// Mitsubishi GX Works2 project: 525252   PLC: Q02/Q02H

PROGRAM MAIN
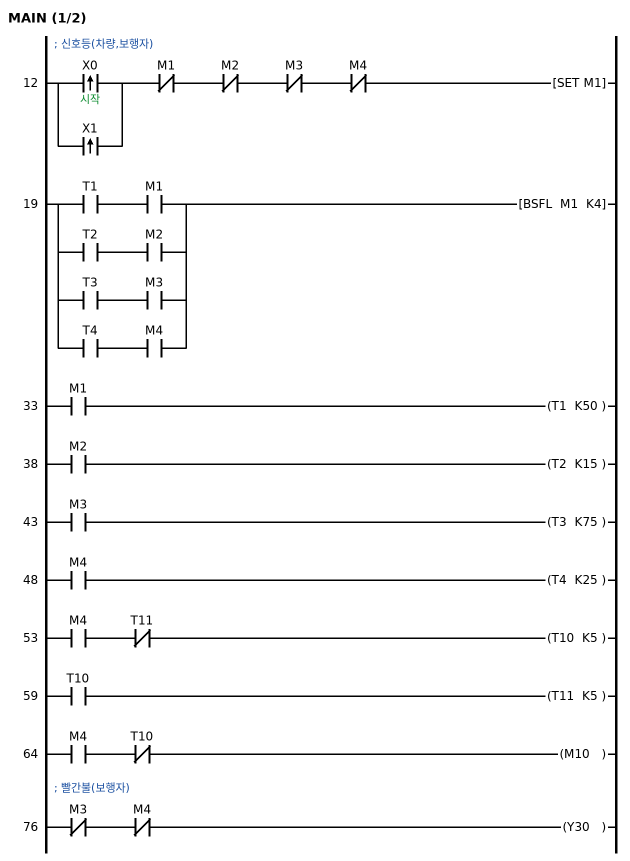
; 신호등(차량,보행자)
12    LDP     X0  ; 시작
      ORP     X1
      ANI     M1
      ANI     M2
      ANI     M3
      ANI     M4
      SET     M1
19    LD      T1
      AND     M1
      LD      T2
      AND     M2
      ORB
      LD      T3
      AND     M3
      ORB
      LD      T4
      AND     M4
      ORB
      BSFL    M1 K4
33    LD      M1
      OUT     T1 K50
38    LD      M2
      OUT     T2 K15
43    LD      M3
      OUT     T3 K75
48    LD      M4
      OUT     T4 K25
53    LD      M4
      ANI     T11
      OUT     T10 K5
59    LD      T10
      OUT     T11 K5
64    LD      M4
      ANI     T10
      OUT     M10
; 빨간불(보행자)
76    LDI     M3
      ANI     M4
      OUT     Y30
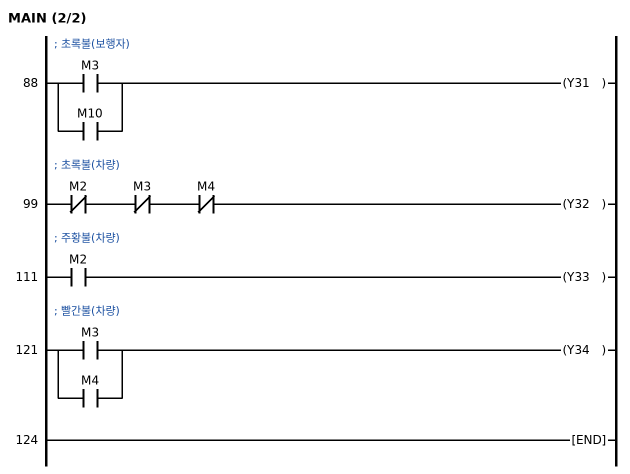
; 초록불(보행자)
88    LD      M3
      OR      M10
      OUT     Y31
; 초록불(차량)
99    LDI     M2
      ANI     M3
      ANI     M4
      OUT     Y32
; 주황불(차량)
111   LD      M2
      OUT     Y33
; 빨간불(차량)
121   LD      M3
      OR      M4
      OUT     Y34
124   END
END_PROGRAM
